// TIA Portal project "conveyer belt system" (V19)

(* hardware
DEVICE "S7-1500/ET200MP station_2"  S7-1500 station
   slot 0: "Rail_0"  Rack  6ES7 590-1***0-0AA0
   slot 1: "PLC_1"  CPU 1515-2 PN  6ES7 515-2AN03-0AB0  V3.0
      slot 3: "CPU display_1"  6ES7591-1BA00-0AA0
      slot 32768: "PROFINET interface_1"  X1
         slot 32769: "Port_1"  X1 P1
         slot 32770: "Port_2"  X1 P2
      slot 33024: "PROFINET interface_2"  X2
         slot 33025: "Port_1"  X2 P1
      slot 34817: "Virtual CP interface port_1"  Virtual CP interface port  Virtual CP interface port
*)

// ===== PLC "PLC_1"  CPU 1515-2 PN =====

VAR_GLOBAL   // PLC tag table "Default tag table"
   "Tag_1" AT %M0.0 : Bool;
   "Tag_2" AT %M1.0 : Bool;
   "Tag_3" AT %M2.0 : Bool;
   "Tag_4" AT %M0.1 : Bool;
   "Tag_5" AT %M0.2 : Bool;
   "Tag_6" AT %M1.1 : Bool;
   "Tag_7" AT %M3.0 : Bool;
END_VAR

VAR_GLOBAL   // PLC tag table "control panel"
   "start button" AT %I0.0 : Bool;
   "reset button" AT %I0.1 : Bool;
   "stop button" AT %I0.2 : Bool;
   "emergency stop" AT %I0.3 : Bool;
   "start button light" AT %Q0.0 : Bool;
   "reset button light" AT %Q0.1 : Bool;
   "stop button light" AT %Q0.2 : Bool;
   "system start" AT %Q0.3 : Bool;
   "system fault" AT %Q0.4 : Bool;
   "system stop" AT %Q0.5 : Bool;
END_VAR

VAR_GLOBAL   // PLC tag table "conveyor 0"
   "motor +" AT %Q3.7 : Bool;
   "motor -" AT %Q3.6 : Bool;
   "encoder A" AT %I2.7 : Bool;
   "encoder B" AT %I2.6 : Bool;
   "sensor" AT %I3.7 : Bool;
END_VAR

VAR_GLOBAL   // PLC tag table "conveyor 1"
   "motor +(1)" AT %Q3.5 : Bool;
   "motor -(1)" AT %Q3.4 : Bool;
   "encoder A(1)" AT %I2.5 : Bool;
   "encoder B(1)" AT %I2.4 : Bool;
   "sensor(1)" AT %I3.6 : Bool;
END_VAR

VAR_GLOBAL   // PLC tag table "conveyor 2"
   "motor +(2)" AT %Q3.3 : Bool;
   "motor -(2)" AT %Q3.2 : Bool;
   "encoder A(2)" AT %I2.2 : Bool;
   "encoder B(2)" AT %I2.3 : Bool;
   "sensor(2)" AT %I3.5 : Bool;
END_VAR

DATA_BLOCK "conveyor 2"   // DB3
{ S7_Optimized_Access := 'TRUE' }
VERSION : 0.1
// stored: InstanceOfName conveyor
"conveyor"
BEGIN
END_DATA_BLOCK

DATA_BLOCK "conveyor 0"   // DB5
{ S7_Optimized_Access := 'TRUE' }
VERSION : 0.1
// stored: InstanceOfName conveyor
"conveyor"
BEGIN
END_DATA_BLOCK

DATA_BLOCK "conveyor 1"   // DB6
{ S7_Optimized_Access := 'TRUE' }
VERSION : 0.1
// stored: InstanceOfName conveyor
"conveyor"
BEGIN
END_DATA_BLOCK

DATA_BLOCK "system start lamp control"   // DB9
{ S7_Optimized_Access := 'TRUE' }
VERSION : 0.1
// stored: InstanceOfName lamp control
"lamp control"
BEGIN
END_DATA_BLOCK

// folder: System blocks/Program resources

DATA_BLOCK "IEC_Timer_0_DB"   // DB1
{ S7_Optimized_Access := 'TRUE' }
AUTHOR : Simatic
FAMILY : IEC
NAME : IEC_TMR
VERSION : 1.0
// stored: InstanceOfName IEC_TIMER
"IEC_TIMER"
BEGIN
END_DATA_BLOCK

DATA_BLOCK "IEC_Timer_0_DB_1"   // DB2
{ S7_Optimized_Access := 'TRUE' }
AUTHOR : Simatic
FAMILY : IEC
NAME : IEC_TMR
VERSION : 1.0
// stored: InstanceOfName IEC_TIMER
"IEC_TIMER"
BEGIN
END_DATA_BLOCK

DATA_BLOCK "IEC_Timer_0_DB_2"   // DB4
{ S7_Optimized_Access := 'TRUE' }
AUTHOR : Simatic
FAMILY : IEC
NAME : IEC_TMR
VERSION : 1.0
// stored: InstanceOfName IEC_TIMER
"IEC_TIMER"
BEGIN
END_DATA_BLOCK

DATA_BLOCK "IEC_Timer_0_DB_3"   // DB7
{ S7_Optimized_Access := 'TRUE' }
AUTHOR : Simatic
FAMILY : IEC
NAME : IEC_TMR
VERSION : 1.0
// stored: InstanceOfName IEC_TIMER
"IEC_TIMER"
BEGIN
END_DATA_BLOCK

DATA_BLOCK "IEC_Timer_0_DB_4"   // DB8
{ S7_Optimized_Access := 'TRUE' }
AUTHOR : Simatic
FAMILY : IEC
NAME : IEC_TMR
VERSION : 1.0
// stored: InstanceOfName IEC_TIMER
"IEC_TIMER"
BEGIN
END_DATA_BLOCK

DATA_BLOCK "IEC_Timer_0_DB_5"   // DB10
{ S7_Optimized_Access := 'TRUE' }
AUTHOR : Simatic
FAMILY : IEC
NAME : IEC_TMR
VERSION : 1.0
// stored: InstanceOfName IEC_TIMER
"IEC_TIMER"
BEGIN
END_DATA_BLOCK

DATA_BLOCK "IEC_Timer_0_DB_6"   // DB11
{ S7_Optimized_Access := 'TRUE' }
AUTHOR : Simatic
FAMILY : IEC
NAME : IEC_TMR
VERSION : 1.0
// stored: InstanceOfName IEC_TIMER
"IEC_TIMER"
BEGIN
END_DATA_BLOCK

// folder: (top level)

FUNCTION_BLOCK "conveyor"   // FB1, LAD
{ S7_Optimized_Access := 'TRUE' }
VERSION : 0.1
   VAR_INPUT
      enable : Bool;
      "encoder A" : Bool;
      "encoder B" : Bool;
      sensor : Bool;
      "preceeding sensor" : Bool;
      "emergency stop" : Bool;
      "clearance time" : Time := T#500MS;
   END_VAR
   VAR_OUTPUT
      "running feedback" : Bool;
      "motor +" : Bool;
      "motor -" : Bool;
   END_VAR
   VAR
      IEC_Timer_0_Instance : TOF_TIME;
      IEC_Timer_0_Instance_1 : TOF_TIME;
      IEC_Timer_0_Instance_2 : TOF_TIME;
      IEC_Timer_0_Instance_3 : TON_TIME;
      "SR latch 1" : Bool;
   END_VAR
BEGIN

REGION Network 1
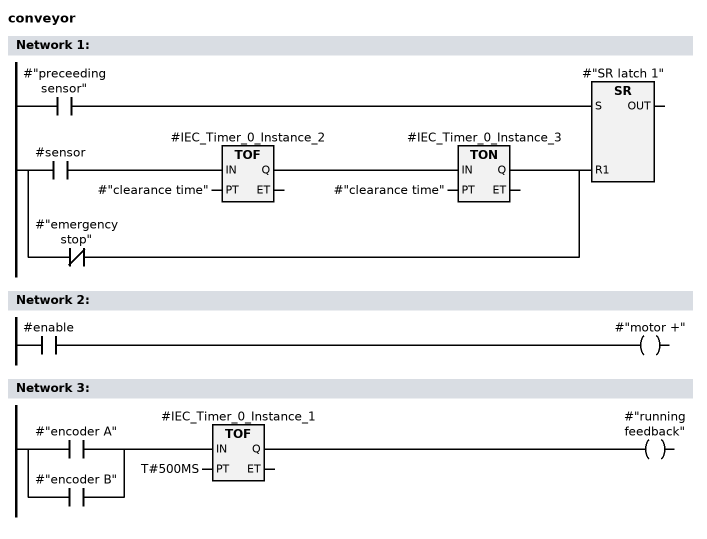
   #IEC_Timer_0_Instance_2(IN := #sensor, PT := #"clearance time");   // TOF
   #IEC_Timer_0_Instance_3(IN := #IEC_Timer_0_Instance_2.Q, PT := #"clearance time");   // TON
   IF #"preceeding sensor" THEN
       #"SR latch 1" := TRUE;   // SR flip-flop
   END_IF;
   IF #IEC_Timer_0_Instance_3.Q OR NOT #"emergency stop" THEN #"SR latch 1" := FALSE; END_IF;
END_REGION

REGION Network 2
   RUNG wire#powerrail
      Contact( #enable )
      Coil( #"motor +" )
   END_RUNG
   // the same network as SCL:
   #"motor +" := #enable;
END_REGION

REGION Network 3
   #IEC_Timer_0_Instance_1(IN := #"encoder A" OR #"encoder B", PT := T#500MS);   // TOF
   #"running feedback" := #IEC_Timer_0_Instance_1.Q;
END_REGION
END_FUNCTION_BLOCK

FUNCTION_BLOCK "lamp control"   // FB2, LAD
{ S7_Optimized_Access := 'TRUE' }
VERSION : 0.1
   VAR_INPUT
      pulse : Bool;
      "pulse time" : Time := T#500MS;
   END_VAR
   VAR_OUTPUT
      "lamp output" : Bool;
   END_VAR
   VAR
      "time delay bit" : Bool;
   END_VAR
BEGIN

REGION Network 1
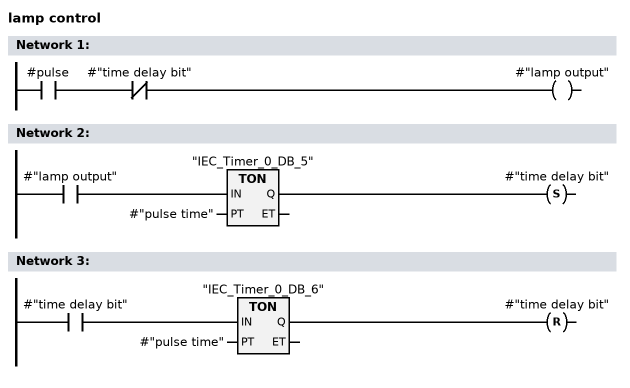
   RUNG wire#powerrail
      Contact( #pulse )
      I_Contact( #"time delay bit" )
      Coil( #"lamp output" )
   END_RUNG
   // the same network as SCL:
   #"lamp output" := #pulse AND NOT #"time delay bit";
END_REGION

REGION Network 2
   "IEC_Timer_0_DB_5".TON(IN := #"lamp output", PT := #"pulse time");
   IF "IEC_Timer_0_DB_5".Q THEN #"time delay bit" := TRUE; END_IF;
END_REGION

REGION Network 3
   "IEC_Timer_0_DB_6".TON(IN := #"time delay bit", PT := #"pulse time");
   IF "IEC_Timer_0_DB_6".Q THEN #"time delay bit" := FALSE; END_IF;
END_REGION
END_FUNCTION_BLOCK

ORGANIZATION_BLOCK "Main"   // OB1, LAD, ProgramCycle
TITLE = "Main Program Sweep (Cycle)"
{ S7_Optimized_Access := 'TRUE' }
VERSION : 0.1
   VAR_INPUT
      Initial_Call : Bool;   // Initial call of this OB
      Remanence : Bool;   // =True, if remanent data are available
   END_VAR
   VAR_TEMP
      "start 1" : Bool;
      "start 2" : Bool;
      "motor 0 enable" : Bool;
      "motor 0 feedback" : Bool;
      "sensor 0 feedback" : Bool;
      "motor 1 enable" : Bool;
      "motor 1 feedback" : Bool;
      "sensor 1 feedback" : Bool;
      "motor 2 enable" : Bool;
      "motor 2 feedback" : Bool;
      "sensor 2 feedback" : Bool;
   END_VAR
   VAR CONSTANT
      "conveyor clear time" : Time;
   END_VAR
BEGIN

REGION Network 1
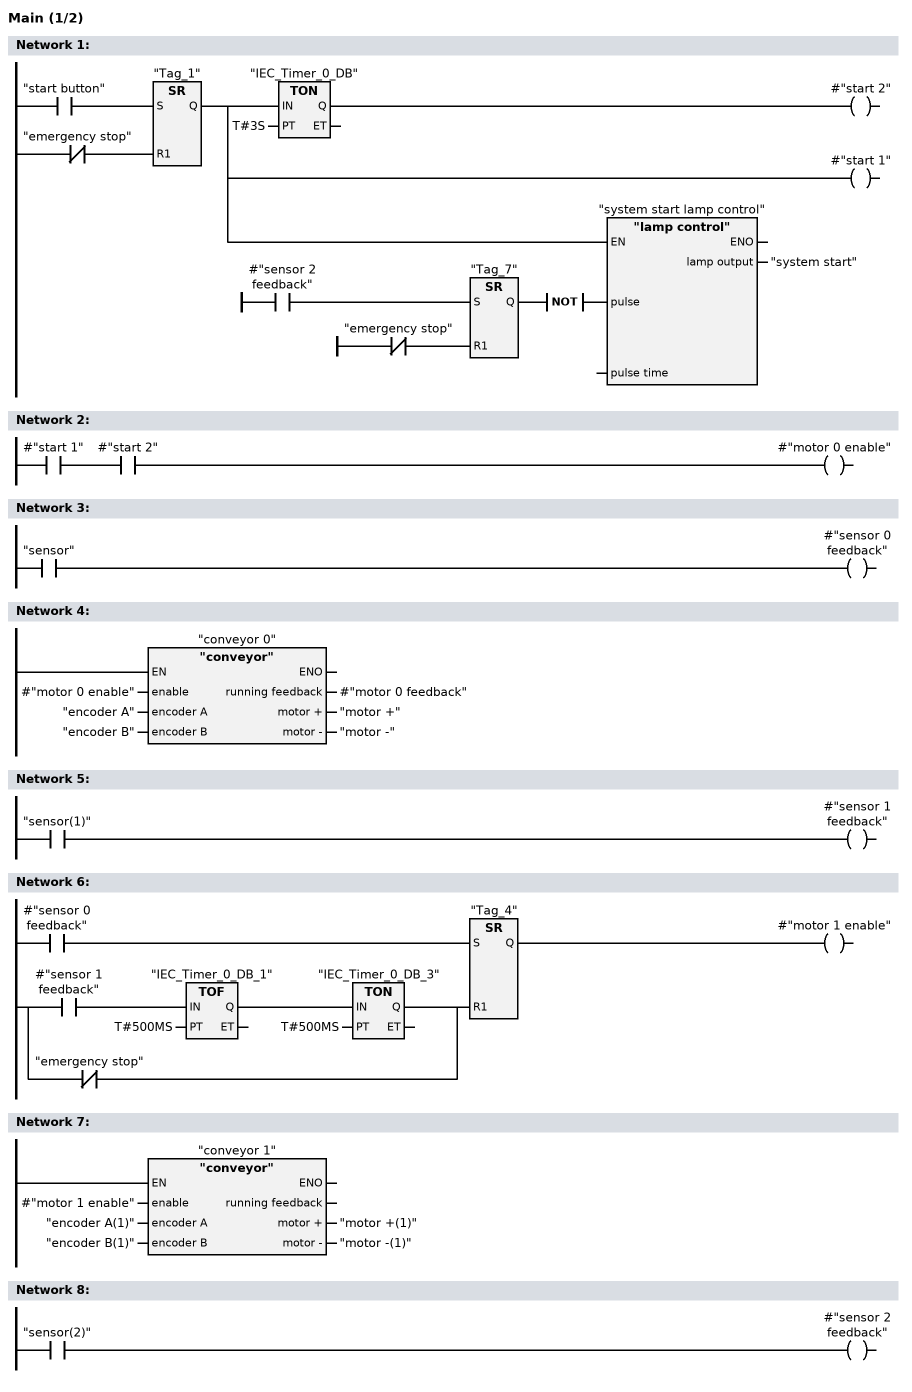
   IF "start button" THEN
       "Tag_1" := TRUE;   // SR flip-flop
   END_IF;
   IF NOT "emergency stop" THEN "Tag_1" := FALSE; END_IF;
   "IEC_Timer_0_DB".TON(IN := "Tag_1", PT := T#3S);
   #"start 2" := "IEC_Timer_0_DB".Q;
   #"start 1" := "Tag_1";
   IF #"sensor 2 feedback" THEN
       "Tag_7" := TRUE;   // SR flip-flop
   END_IF;
   IF NOT "emergency stop" THEN "Tag_7" := FALSE; END_IF;
   IF "Tag_1" THEN
       "system start lamp control"(pulse := NOT "Tag_7", "lamp output" => "system start");   // "lamp control"
   END_IF;
END_REGION

REGION Network 2
   RUNG wire#powerrail
      Contact( #"start 1" )
      Contact( #"start 2" )
      Coil( #"motor 0 enable" )
   END_RUNG
   // the same network as SCL:
   #"motor 0 enable" := #"start 1" AND #"start 2";
END_REGION

REGION Network 3
   RUNG wire#powerrail
      Contact( "sensor" )
      Coil( #"sensor 0 feedback" )
   END_RUNG
   // the same network as SCL:
   #"sensor 0 feedback" := "sensor";
END_REGION

REGION Network 4
   RUNG wire#powerrail
      "conveyor 0"(enable := #"motor 0 enable", "encoder A" := "encoder A", "encoder B" := "encoder B", "running feedback" => #"motor 0 feedback", "motor +" => "motor +", "motor -" => "motor -")
   END_RUNG
   // the same network as SCL:
   "conveyor 0"(enable := #"motor 0 enable",   // "conveyor"
                "encoder A" := "encoder A",
                "encoder B" := "encoder B",
                "running feedback" => #"motor 0 feedback",
                "motor +" => "motor +",
                "motor -" => "motor -");
END_REGION

REGION Network 5
   RUNG wire#powerrail
      Contact( "sensor(1)" )
      Coil( #"sensor 1 feedback" )
   END_RUNG
   // the same network as SCL:
   #"sensor 1 feedback" := "sensor(1)";
END_REGION

REGION Network 6
   "IEC_Timer_0_DB_1".TOF(IN := #"sensor 1 feedback", PT := T#500MS);
   "IEC_Timer_0_DB_3".TON(IN := "IEC_Timer_0_DB_1".Q, PT := T#500MS);
   IF #"sensor 0 feedback" THEN
       "Tag_4" := TRUE;   // SR flip-flop
   END_IF;
   IF "IEC_Timer_0_DB_3".Q OR NOT "emergency stop" THEN "Tag_4" := FALSE; END_IF;
   #"motor 1 enable" := "Tag_4";
END_REGION

REGION Network 7
   RUNG wire#powerrail
      "conveyor 1"(enable := #"motor 1 enable", "encoder A" := "encoder A(1)", "encoder B" := "encoder B(1)", "running feedback" =>, "motor +" => "motor +(1)", "motor -" => "motor -(1)")
   END_RUNG
   // the same network as SCL:
   "conveyor 1"(enable := #"motor 1 enable",   // "conveyor"
                "encoder A" := "encoder A(1)",
                "encoder B" := "encoder B(1)",
                "motor +" => "motor +(1)",
                "motor -" => "motor -(1)");
END_REGION

REGION Network 8
   RUNG wire#powerrail
      Contact( "sensor(2)" )
      Coil( #"sensor 2 feedback" )
   END_RUNG
   // the same network as SCL:
   #"sensor 2 feedback" := "sensor(2)";
END_REGION

REGION Network 9
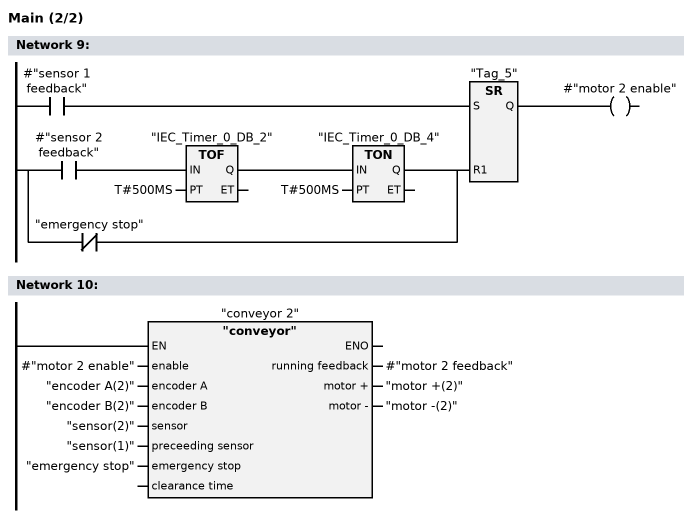
   "IEC_Timer_0_DB_2".TOF(IN := #"sensor 2 feedback", PT := T#500MS);
   "IEC_Timer_0_DB_4".TON(IN := "IEC_Timer_0_DB_2".Q, PT := T#500MS);
   IF #"sensor 1 feedback" THEN
       "Tag_5" := TRUE;   // SR flip-flop
   END_IF;
   IF "IEC_Timer_0_DB_4".Q OR NOT "emergency stop" THEN "Tag_5" := FALSE; END_IF;
   #"motor 2 enable" := "Tag_5";
END_REGION

REGION Network 10
   RUNG wire#powerrail
      "conveyor 2"(enable := #"motor 2 enable", "encoder A" := "encoder A(2)", "encoder B" := "encoder B(2)", sensor := "sensor(2)", "preceeding sensor" := "sensor(1)", "emergency stop" := "emergency stop", "clearance time" :=, "running feedback" => #"motor 2 feedback", "motor +" => "motor +(2)", "motor -" => "motor -(2)")
   END_RUNG
   // the same network as SCL:
   "conveyor 2"(enable := #"motor 2 enable",   // "conveyor"
                "encoder A" := "encoder A(2)",
                "encoder B" := "encoder B(2)",
                sensor := "sensor(2)",
                "preceeding sensor" := "sensor(1)",
                "emergency stop" := "emergency stop",
                "running feedback" => #"motor 2 feedback",
                "motor +" => "motor +(2)",
                "motor -" => "motor -(2)");
END_REGION
END_ORGANIZATION_BLOCK